// Mitsubishi GX Works2 project: nuclear   PLC: FX3U/FX3UC

PROGRAM MAIN
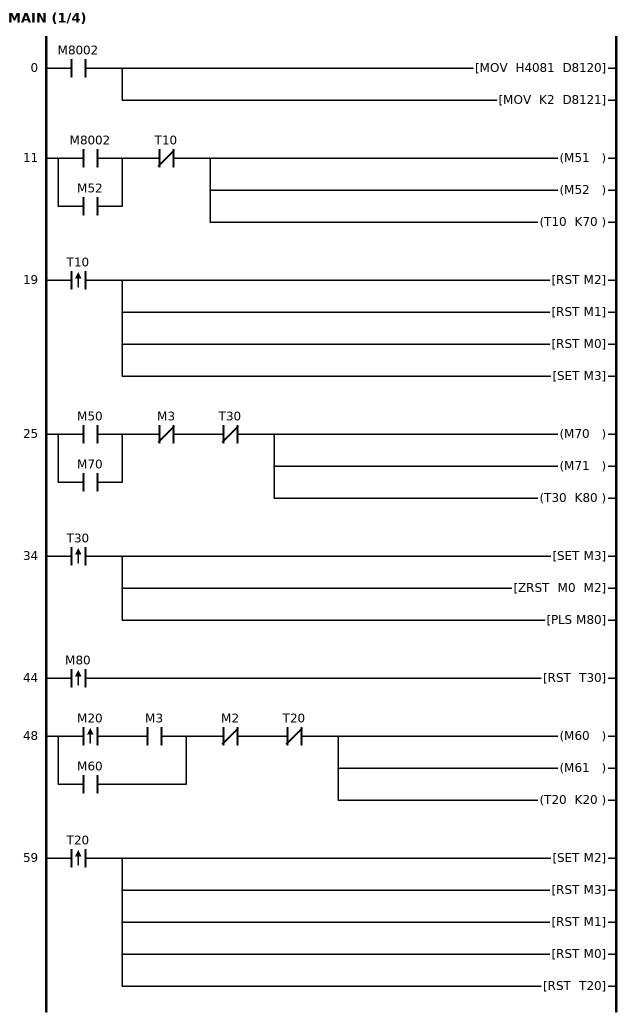
0     LD      M8002
      MOV     H4081 D8120
      MOV     K2 D8121
11    LD      M8002
      OR      M52
      ANI     T10
      OUT     M51
      OUT     M52
      OUT     T10 K70
19    LDP     T10
      RST     M2
      RST     M1
      RST     M0
      SET     M3
25    LD      M50
      OR      M70
      ANI     M3
      ANI     T30
      OUT     M70
      OUT     M71
      OUT     T30 K80
34    LDP     T30
      SET     M3
      ZRST    M0 M2
      PLS     M80
44    LDP     M80
      RST     T30
48    LDP     M20
      AND     M3
      OR      M60
      ANI     M2
      ANI     T20
      OUT     M60
      OUT     M61
      OUT     T20 K20
59    LDP     T20
      SET     M2
      RST     M3
      RST     M1
      RST     M0
      RST     T20
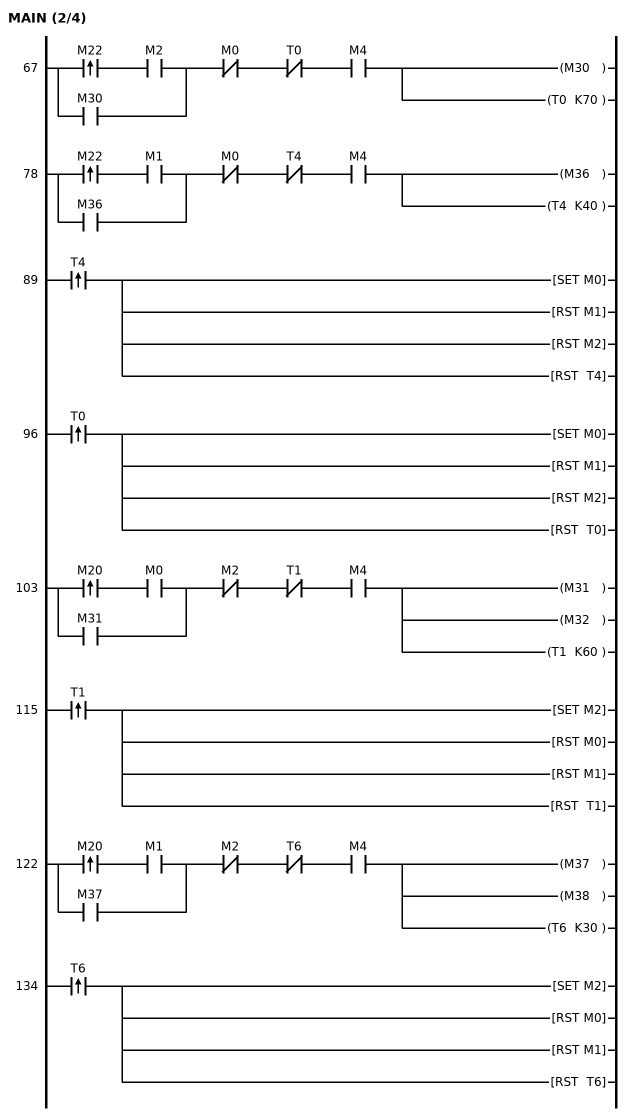
67    LDP     M22
      AND     M2
      OR      M30
      ANI     M0
      ANI     T0
      AND     M4
      OUT     M30
      OUT     T0 K70
78    LDP     M22
      AND     M1
      OR      M36
      ANI     M0
      ANI     T4
      AND     M4
      OUT     M36
      OUT     T4 K40
89    LDP     T4
      SET     M0
      RST     M1
      RST     M2
      RST     T4
96    LDP     T0
      SET     M0
      RST     M1
      RST     M2
      RST     T0
103   LDP     M20
      AND     M0
      OR      M31
      ANI     M2
      ANI     T1
      AND     M4
      OUT     M31
      OUT     M32
      OUT     T1 K60
115   LDP     T1
      SET     M2
      RST     M0
      RST     M1
      RST     T1
122   LDP     M20
      AND     M1
      OR      M37
      ANI     M2
      ANI     T6
      AND     M4
      OUT     M37
      OUT     M38
      OUT     T6 K30
134   LDP     T6
      SET     M2
      RST     M0
      RST     M1
      RST     T6
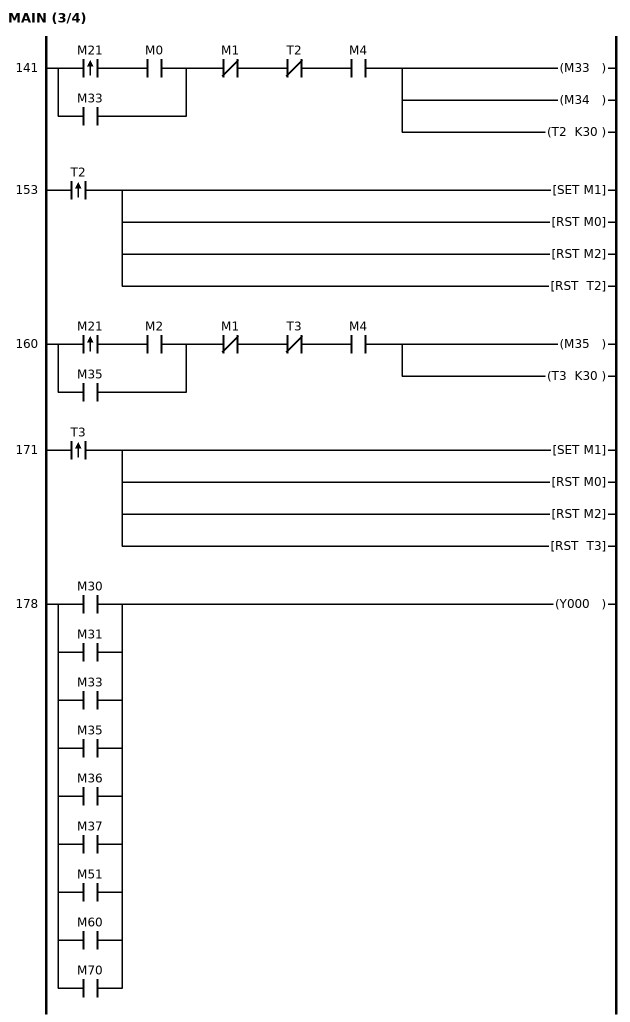
141   LDP     M21
      AND     M0
      OR      M33
      ANI     M1
      ANI     T2
      AND     M4
      OUT     M33
      OUT     M34
      OUT     T2 K30
153   LDP     T2
      SET     M1
      RST     M0
      RST     M2
      RST     T2
160   LDP     M21
      AND     M2
      OR      M35
      ANI     M1
      ANI     T3
      AND     M4
      OUT     M35
      OUT     T3 K30
171   LDP     T3
      SET     M1
      RST     M0
      RST     M2
      RST     T3
178   LD      M30
      OR      M31
      OR      M33
      OR      M35
      OR      M36
      OR      M37
      OR      M51
      OR      M60
      OR      M70
      OUT     Y000
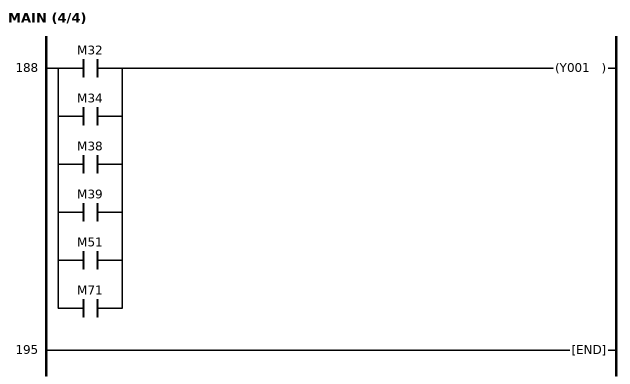
188   LD      M32
      OR      M34
      OR      M38
      OR      M39
      OR      M51
      OR      M71
      OUT     Y001
195   END
END_PROGRAM
